Universal Robots PolyScope program: Dovetail_top.urp

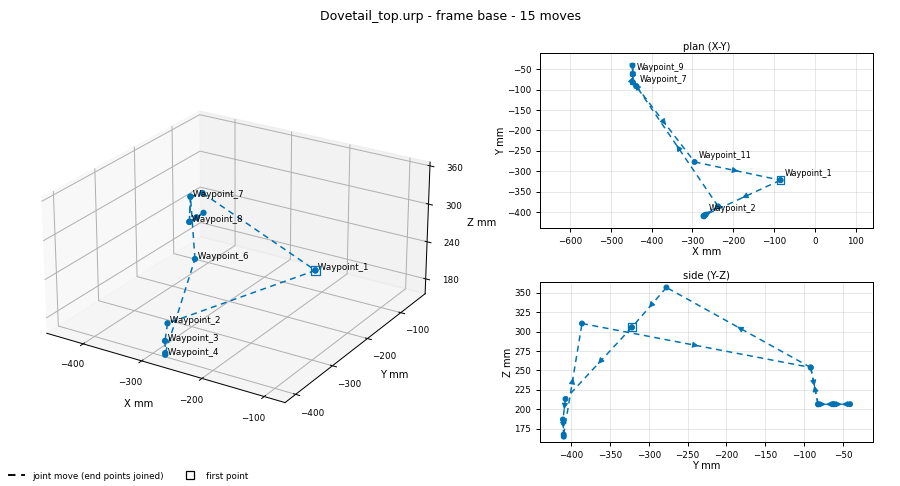
[picture p0: tool path of Dovetail_top.urp in frame base, 15 of 15 moves have a stored position in this frame; points joined in program order, loops and branches not executed]
Program Dovetail_top (installation=default directory=/programs/usbdisk/Zahra1/orangi createdIn=5.11.11.1010533 lastSavedIn=5.11.11.1010533 robotSerialNumber=20205300864)
Calibrated DH parameters: a=[-0.000166, -0.243494, -0.153108, 0.000057, -0.000123, 0]; d=[0.151897, -1.34267, 53.988124, -52.514559, 0.085283, 0.092193]; alpha=[1.572472, -0.003756, 0.002824, 1.570807, -1.572621, 0]; deltaTheta=[0, 0.020704, 7.033215, -0.770746, 0.000004, 0]
Robot Program (runOnlyOnce=true)
  MoveJ speed 60 deg/s, acceleration 80 deg/s^2 (useActiveTCP=true) feature=Base
    Waypoint Waypoint_1: TCP in base x=-84.299 y=-321.875 z=305.481 mm, rx=-2.0809 ry=-2.2572 rz=0.0984 rad; joints [-79.978, -91.201, -87.971, -91.7, 84.671, 815.506] deg
    URCap Gripper (Robotiq_Grippers, Robotiq Inc.) dataModel(position=40.3921568627451, force=97.0, speed=52.0, positionInDouble=40.3921568627451, forceInDouble=97.0, speedInDouble=52.0, slaveIds=[9], blocking=true, robotCompliant=false)
    Waypoint Waypoint_2: TCP in base x=-269.534 y=-407.293 z=213.302 mm, rx=-3.0931 ry=0.1111 rz=0.0835 rad; joints [-107.274, -135.459, -48.529, -87.612, 86.216, 886.941] deg
    Waypoint Waypoint_3: TCP in base x=-271.882 y=-410.512 z=186.915 mm, rx=-3.0931 ry=0.0735 rz=0.0514 rad; joints [-107.649, -137.957, -50.912, -83.09, 87.297, 885.175] deg
    Waypoint Waypoint_4: TCP in base x=-272.588 y=-409.473 z=164.766 mm, rx=-3.0933 ry=0.0735 rz=0.0514 rad; joints [-107.778, -139.101, -54.846, -77.995, 87.3, 885.052] deg
    URCap Gripper (Robotiq_Grippers, Robotiq Inc.) dataModel(position=75.01960784313725, force=97.0, speed=52.0, positionInDouble=75.01960784313725, forceInDouble=97.0, speedInDouble=52.0, slaveIds=[9], blocking=true, robotCompliant=false)
    Waypoint Waypoint_5: TCP in base x=-272.516 y=-409.599 z=167.547 mm, rx=-3.0934 ry=0.0735 rz=0.0514 rad; joints [-107.764, -138.93, -54.401, -78.609, 87.301, 885.065] deg
    Waypoint Waypoint_6: TCP in base x=-237.115 y=-386.022 z=310.438 mm, rx=3.1293 ry=0.0114 rz=-0.0767 rad; joints [-104.239, -124.25, -42.915, -101.405, 87.317, 885.35] deg
    Waypoint Waypoint_7: TCP in base x=-437.484 y=-91.575 z=253.815 mm, rx=-3.1095 ry=0.0382 rz=0.0804 rad; joints [-150.558, -120.969, -63.707, -83.546, 86.905, 840.881] deg
    Waypoint Waypoint_8: TCP in base x=-446.275 y=-82.057 z=206.473 mm, rx=-3.0272 ry=0.0204 rz=-0.0482 rad; joints [-151.854, -126.692, -64.692, -83.25, 85.065, 839.207] deg
    Waypoint Waypoint_9: motionParameters(jointSpeed=0.349066 jointAcceleration=0.174533 cartesianSpeed=0.25 cartesianAcceleration=1.2); TCP in base x=-446.268 y=-61.939 z=206.549 mm, rx=-3.0247 ry=0.0227 rz=-0.0549 rad; joints [-154.199, -125.841, -66.083, -82.802, 84.871, 836.961] deg
    Waypoint Waypoint_12: TCP in base x=-446.9 y=-40.958 z=206.606 mm, rx=-3.0881 ry=0.0652 rz=-0.0584 rad; joints [-157.479, -125.195, -67.691, -80.199, 88.06, 835.088] deg
    URCap Gripper (Robotiq_Grippers, Robotiq Inc.) dataModel(position=38.431372549019606, force=97.0, speed=52.0, positionInDouble=38.431372549019606, forceInDouble=97.0, speedInDouble=52.0, slaveIds=[9], blocking=true, robotCompliant=false)
    Waypoint Waypoint_9: motionParameters(jointSpeed=0.349066 jointAcceleration=0.174533 cartesianSpeed=0.25 cartesianAcceleration=1.2); TCP in base x=-446.268 y=-61.939 z=206.549 mm, rx=-3.0247 ry=0.0227 rz=-0.0549 rad; joints [-154.199, -125.841, -66.083, -82.802, 84.871, 836.961] deg
    Waypoint Waypoint_8: TCP in base x=-446.275 y=-82.057 z=206.473 mm, rx=-3.0272 ry=0.0204 rz=-0.0482 rad; joints [-151.854, -126.692, -64.692, -83.25, 85.065, 839.207] deg
    Waypoint Waypoint_7: TCP in base x=-437.484 y=-91.575 z=253.815 mm, rx=-3.1095 ry=0.0382 rz=0.0804 rad; joints [-150.558, -120.969, -63.707, -83.546, 86.905, 840.881] deg
    Waypoint Waypoint_11: TCP in base x=-294.805 y=-277.288 z=356.828 mm, rx=-1.8865 ry=-2.467 rz=-0.0298 rad; joints [-117.454, -114.271, -44.517, -112.545, 88.059, 767.431] deg
    Waypoint Waypoint_1: TCP in base x=-84.299 y=-321.875 z=305.481 mm, rx=-2.0809 ry=-2.2572 rz=0.0984 rad; joints [-79.978, -91.201, -87.971, -91.7, 84.671, 815.506] deg
